Fanuc KAREL source: kt00710.KL

-- PROVISIONAL review KL for V770-1; original PC SHA256 070ca527e66322fc9beb9cfc4eb19756ddb397a91c3b55d926daab394fd1990c
-- Incomplete behavior may be omitted. Consult companion uncertainty JSON. Do not deploy.
PROGRAM KT00710
%NOLOCKGROUP
VAR
  B1 : BOOLEAN
  B2 : BOOLEAN
  OUT : BOOLEAN
BEGIN
  -- UNRESOLVED_PC offsets 5-12; opcodes 9D,23
  -- UNRESOLVED_PC offsets 17-24; opcodes 9C,23
  -- UNRESOLVED_PC offsets 29-36; opcodes 9D,23
  -- UNRESOLVED_PC offsets 41-48; opcodes 9C,23
  -- UNRESOLVED_PC offsets 53-68; opcodes 22,63,23
  -- UNRESOLVED_PC offsets 73-77; opcodes 7F
END KT00710
